INTERFACE IRouteableComponent EXTENDS IACComponent

METHOD AddPoint : BOOL
VAR_INPUT
	point : IACPoint;
END_VAR
END_METHOD

PROPERTY Points : ARRAY [1..GCL.cPointMAX] OF IACPoint
GET
END_GET
END_PROPERTY

END_INTERFACE

(* stored: Version 1.1.0.1, ProductVersion 3.1.4020.12
   Itf IRouteableComponent: Id {1b544dde-b4cf-4e5c-b560-d8ca28cdf1ad}
   Method AddPoint: Id {3c8aa412-f5f3-4530-94da-866888505000}
   Property Points: Id {44b89c15-a05d-424d-8f11-9c8492448fb4}
   Get Get: Id {78ac50a8-605d-4d52-b528-4da5c5de96d1} *)
